FUNCTION_BLOCK FB_PM2200 EXTENDS FB_ModbusSlave
VAR
	arrAccPower	:	ARRAY [0..41] OF WORD;
	arrQuaPower		:	ARRAY [0..17] OF WORD;
	arrCommon		:	ARRAY [0..111] OF WORD;
END_VAR

PROPERTY AccPower : ARRAY [0..41] OF WORD
GET
AccPower := arrAccPower;
END_GET
END_PROPERTY

PROPERTY Common : ARRAY [0..111] OF WORD
GET
Common := arrCommon;
END_GET
END_PROPERTY

METHOD Convert : BOOL
VAR_INPUT
	iRegionNo	:	INT;
	pReadData	:	POINTER TO BYTE;
END_VAR
VAR
	pTempData	: 	POINTER TO BYTE;
	iTempData	: 	BYTE;
	iLoop		: 	INT;
	bHiByte		:	BOOL := TRUE;
END_VAR
CASE iRegionNo OF
	0: 
		FOR iLoop := 0 TO SIZEOF(arrAccPower)*2 DO
			pTempData := (pReadData + iLoop);
			iTempData := pTempData^;
			
			IF bHiByte THEN
				arrAccPower[iLoop/2] := SHL(BYTE_TO_WORD(iTempData), 8);
			ELSE 
				arrAccPower[iLoop/2] := arrAccPower[iLoop/2] + BYTE_TO_WORD(iTempData);
				IF bSwap THEN
					arrAccPower[iLoop/2] := ROL(arrAccPower[iLoop/2], 8);
				END_IF
			END_IF
			bHiByte := NOT bHiByte;
		END_FOR
		
	1: 
		FOR iLoop := 0 TO SIZEOF(arrQuaPower)*2 DO
			pTempData := (pReadData + iLoop);
			iTempData := pTempData^;
			
			IF bHiByte THEN
				arrQuaPower[iLoop/2] := SHL(BYTE_TO_WORD(iTempData), 8);
			ELSE 
				arrQuaPower[iLoop/2] := arrQuaPower[iLoop/2] + BYTE_TO_WORD(iTempData);
				IF bSwap THEN
					arrQuaPower[iLoop/2] := ROL(arrQuaPower[iLoop/2], 8);
				END_IF
			END_IF
			bHiByte := NOT bHiByte;
		END_FOR

	2: 
		FOR iLoop := 0 TO SIZEOF(arrCommon)*2 DO
			pTempData := (pReadData + iLoop);
			iTempData := pTempData^;
			
			IF bHiByte THEN
				arrCommon[iLoop/2] := SHL(BYTE_TO_WORD(iTempData), 8);
			ELSE 
				arrCommon[iLoop/2] := arrCommon[iLoop/2] + BYTE_TO_WORD(iTempData);
				IF bSwap THEN
					arrCommon[iLoop/2] := ROL(arrCommon[iLoop/2], 8);
				END_IF
			END_IF
			bHiByte := NOT bHiByte;
		END_FOR

END_CASE
END_METHOD

METHOD FirstCycle : BOOL
VAR_INPUT
END_VAR
arrAddress[0][0] := 2999;			// Current
arrAddress[0][1] := 12;

arrAddress[1][0] := 3019;			// Voltage
arrAddress[1][1] := 14;		
		
arrAddress[2][0] := 3053;
arrAddress[2][1] := 16;				// Power
arrAddress[3][0] := 3069;
arrAddress[3][1] := 8;				

arrAddress[4][0] := 3077;			// Power factor
arrAddress[4][1] := 16;		
		
arrAddress[5][0] := 3109;			// Frequency
arrAddress[6][1] := 2;				

iNumAddRegion := 6;
END_METHOD

PROPERTY QuaPower : ARRAY [0..17] OF WORD
GET
QuaPower := arrQuaPower;
END_GET
END_PROPERTY

END_FUNCTION_BLOCK

(* stored: Version 1.1.0.1, ProductVersion 3.1.4024.12
   POU FB_PM2200: Id {424297d8-0415-4cca-806d-7c8a11b0f60c}, SpecialFunc None
   Property AccPower: Id {511a922c-16b5-40eb-b342-f003d5c054a8}
   Get Get: Id {35dbaf46-f127-4597-b6d3-dce96a332af9}
   Property Common: Id {01ab0b79-be49-4632-92d6-b78b627ca829}
   Get Get: Id {16e0c163-60d1-404e-9068-65d270bfe7d7}
   Method Convert: Id {276333c7-3466-47b5-afde-518a7f2664a8}
   Method FirstCycle: Id {e08c1b98-7f51-4715-953e-b416f51dff4f}
   Property QuaPower: Id {2a9e310c-a3ac-4af1-b587-dbdf2f800895}
   Get Get: Id {a45de528-117b-4c7c-9bf5-dc69edceaf41} *)
